// TIA Portal V20 export
DATA_BLOCK "DB_DigitalInputs"   // DB2210
// stored: AutoNumber false, InstanceOfName FB_DigitalInputs, InstanceOfType FB
"FB_DigitalInputs"
   // VAR
   //    sFreeI0_0 : "FB_DigitalInput";
   //    sX_AxisBrakePressCtrl : "FB_DigitalInput";
   //    sY_AxisBrakePressCtrl : "FB_DigitalInput";
   //    sBreakerCtrl : "FB_DigitalInput";
   //    sCabinetTemperatureCtrl : "FB_DigitalInput";
   //    sUPS_PowerFailure : "FB_DigitalInput";
   //    sAirPressureCtrl : "FB_DigitalInput";
   //    sShutterClosed : "FB_DigitalInput";
   //    sAirDryerOK : "FB_DigitalInput";
   //    sUPS_BatteryOK : "FB_DigitalInput";
   //    sFrontDoorClosed : "FB_DigitalInput";
   //    sInfeedReadyOK_Start : "FB_DigitalInput";
   //    sCoolingOK : "FB_DigitalInput";
   //    sFreeI1_5 : "FB_DigitalInput";
   //    sPowerReady : "FB_DigitalInput";
   //    sAlarmI2T : "FB_DigitalInput";
   //    sHeadLaserBusy : "FB_DigitalInput";
   //    sHeadLaserBreaker { S7_SetPoint := 'True'} : "FB_DigitalInput";
   //    sFrontDoorLocked { S7_SetPoint := 'True'} : "FB_DigitalInput";
   //    sUPS_CommonAlarm { S7_SetPoint := 'True'} : "FB_DigitalInput";
   //    sUPS_BatteryLow { S7_SetPoint := 'True'} : "FB_DigitalInput";
   //    sFreeI2_5 { S7_SetPoint := 'True'} : "FB_DigitalInput";
   //    sHeadChillerHighPressure { S7_SetPoint := 'True'} : "FB_DigitalInput";
   //    sHeadChillerWaterTemperature { S7_SetPoint := 'True'} : "FB_DigitalInput";
   //    sHeadChillerFlow { S7_SetPoint := 'True'} : "FB_DigitalInput";
   //    sHeadChillerCollectivFault { S7_SetPoint := 'True'} : "FB_DigitalInput";
   //    sHeadChillerWaterLevel { S7_SetPoint := 'True'} : "FB_DigitalInput";
   //    sUPS_ByPassActive { S7_SetPoint := 'True'} : "FB_DigitalInput";
   //    sHeadChillerAmbiantTemperature { S7_SetPoint := 'True'} : "FB_DigitalInput";
   //    sFreeI3_5 { S7_SetPoint := 'True'} : "FB_DigitalInput";
   //    sFreeI3_6 { S7_SetPoint := 'True'} : "FB_DigitalInput";
   //    sFreeI3_7 { S7_SetPoint := 'True'} : "FB_DigitalInput";
   //    sLoadClampOpened { S7_SetPoint := 'True'} : "FB_DigitalInput";
   //    sLoadClampNotClosedWithPart { S7_SetPoint := 'True'} : "FB_DigitalInput";
   //    sUnloadClampOpened { S7_SetPoint := 'True'} : "FB_DigitalInput";
   //    sUPS_Fault { S7_SetPoint := 'True'} : "FB_DigitalInput";
   //    sInternalGateLocked { S7_SetPoint := 'True'} : "FB_DigitalInput";
   //    sExternalGateLocked { S7_SetPoint := 'True'} : "FB_DigitalInput";
   //    sInverterActive { S7_SetPoint := 'True'} : "FB_DigitalInput";
   //    sUnloadClampNotClosedWithPart { S7_SetPoint := 'True'} : "FB_DigitalInput";
   //    sFreeI5_0 { S7_SetPoint := 'True'} : "FB_DigitalInput";
   //    sFreeI5_1 { S7_SetPoint := 'True'} : "FB_DigitalInput";
   //    sInternalGateOpened { S7_SetPoint := 'True'} : "FB_DigitalInput";
   //    sExternalGateOpened { S7_SetPoint := 'True'} : "FB_DigitalInput";
   //    sPowerMeterBackCtrl { S7_SetPoint := 'True'} : "FB_DigitalInput";
   //    sPowerMeterFrontCtrl { S7_SetPoint := 'True'} : "FB_DigitalInput";
   //    sFreeI5_6 { S7_SetPoint := 'True'} : "FB_DigitalInput";
   //    sFreeI5_7 { S7_SetPoint := 'True'} : "FB_DigitalInput";
   //    sHeadChillerCutOff { S7_SetPoint := 'True'} : "FB_DigitalInput";
   //    sHeadChillerTemperature { S7_SetPoint := 'True'} : "FB_DigitalInput";
   //    sFreeI6_2 { S7_SetPoint := 'True'} : "FB_DigitalInput";
   //    sFreeI6_3 { S7_SetPoint := 'True'} : "FB_DigitalInput";
   //    sClampingOpenCtrl { S7_SetPoint := 'True'} : "FB_DigitalInput";
   //    sB_Axis_BrakeReleasedCtrl { S7_SetPoint := 'True'} : "FB_DigitalInput";
   //    sFreeI6_6 { S7_SetPoint := 'True'} : "FB_DigitalInput";
   //    sB_AxisReferencePoint { S7_SetPoint := 'True'} : "FB_DigitalInput";
   //    sSourceChillerHighPressure { S7_SetPoint := 'True'} : "FB_DigitalInput";
   //    sSourceChillerWaterTemperature { S7_SetPoint := 'True'} : "FB_DigitalInput";
   //    sSourceChillerFlow { S7_SetPoint := 'True'} : "FB_DigitalInput";
   //    sSourceChillerCollectivFault { S7_SetPoint := 'True'} : "FB_DigitalInput";
   //    sSourceChillerWaterLevel { S7_SetPoint := 'True'} : "FB_DigitalInput";
   //    sSourceChillerAmbiantTemperature { S7_SetPoint := 'True'} : "FB_DigitalInput";
   //    sSourceChillerCutOff { S7_SetPoint := 'True'} : "FB_DigitalInput";
   //    sSourceChillerTemperature { S7_SetPoint := 'True'} : "FB_DigitalInput";
   // END_VAR
BEGIN
END_DATA_BLOCK
